FUNCTION_BLOCK fb_LocalTime
VAR_INPUT

END_VAR
VAR_OUTPUT
  sLocalTime  : STRING;
  dtLocalTime : DT;
END_VAR
VAR
  GetSysTime    : FW_GetSystemTime;
  strFileTime   : Tc2_Utilities.T_FILETIME;
END_VAR

GetSysTime(dwTimeLo=> strFileTime.dwLowDateTime, dwTimeHi=> strFileTime.dwHighDateTime);

sLocalTime := SYSTEMTIME_TO_STRING( FILETIME_TO_SYSTEMTIME( strFileTime ) );
dtLocalTime := systemtime_to_dt( FILETIME_TO_SYSTEMTIME( strFileTime ) );

END_FUNCTION_BLOCK

(* stored: Version 1.1.0.1, ProductVersion 3.1.4024.9
   POU fb_LocalTime: Id {4d26523e-7cf5-060f-2676-dd94d0395994}, SpecialFunc None *)
